(* IEC 61131-3 sources: GP-Electronics/assets/projects/plc-mvp, 1 file *)

(* ---- blink.st ---- *)
PROGRAM Blink
VAR
  out1: BOOL;
  count: INT;
END_VAR

out1 := TRUE;
count := 42;
END_PROGRAM
